Omron CX-Programmer project NewProject (CX-Programmer 9.73)

# PLC PLC_Traffic_Lights: CP1E E20

## Global symbols (name address type ; comment)
0.00 BOOL  ; START
0.01 BOOL  ; STOP
100.00 BOOL  ; LAMPU HIJAU SIMPANG 1
100.01 BOOL  ; LAMPU KUNING SIMPANG 1
100.02 BOOL  ; LAMPU MERAH SIMPANG 1
100.03 BOOL  ; LAMPU HIJAU SIMPANG 2
100.04 BOOL  ; LAMPU KUNING SIMPANG 2
100.05 BOOL  ; LAMPU MERAH SIMPANG 2
100.06 BOOL  ; LAMPU HIJAU SIMPANG 3
100.07 BOOL  ; LAMPU KUNING SIMPANG 3
100.08 BOOL  ; LAMPU MERAH SIMPANG 3
100.09 BOOL  ; LAMPU HIJAU SIMPANG 4
100.10 BOOL  ; LAMPU KUNING SIMPANG 4
100.11 BOOL  ; LAMPU MERAH SIMPANG 4
100.12 BOOL  ; LAMPU PEJALAN KAKI MERAH 1
100.13 BOOL  ; LAMPU PEJALAN KAKI MERAH 2
100.14 BOOL  ; LAMPU PEJALAN KAKI MERAH 3
100.15 BOOL  ; LAMPU PEJALAN KAKI MERAH 4
101.00 BOOL  ; LAMPU PEJALAN KAKI MERAH 1
101.01 BOOL  ; LAMPU PEJALAN KAKI HIJAU 1
101.02 BOOL  ; LAMPU PEJALAN KAKI MERAH 2
101.03 BOOL  ; LAMPU PEJALAN KAKI HIJAU 2
101.04 BOOL  ; LAMPU PEJALAN KAKI MERAH 3
101.05 BOOL  ; LAMPU PEJALAN KAKI HIJAU 3
101.06 BOOL  ; LAMPU PEJALAN KAKI MERAH 3
101.07 BOOL  ; LAMPU PEJALAN KAKI HIJAU 4
99.00 BOOL  ; LAMPU PEJALAN KAKI HIJAU 1
99.01 BOOL  ; LAMPU PEJALAN KAKI HIJAU 2
99.02 BOOL  ; LAMPU PEJALAN KAKI HIJAU 3
99.03 BOOL  ; LAMPU PEJALAN KAKI HIJAU 4
W0.00 BOOL  ; RUNNING

## Program NewProgram1 (cyclic task 0)
; PLC Traffic Lights

### Section Section1

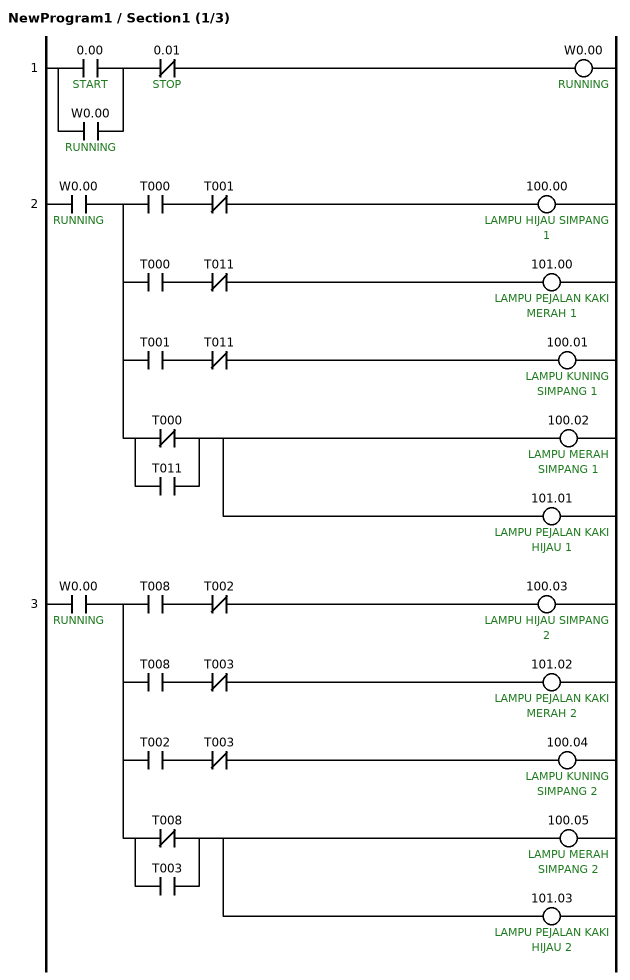
; rung 1
LD 0.00  ; START
OR W0.00  ; RUNNING
ANDNOT 0.01  ; STOP
OUT W0.00  ; RUNNING
; rung 2
LD W0.00  ; RUNNING
OUT TR0
AND T000
ANDNOT T001
OUT 100.00  ; LAMPU HIJAU SIMPANG 1
LD TR0
AND T000
ANDNOT T011
OUT 101.00  ; LAMPU PEJALAN KAKI MERAH 1
LD TR0
AND T001
ANDNOT T011
OUT 100.01  ; LAMPU KUNING SIMPANG 1
LD TR0
LDNOT T000
OR T011
ANDLD
OUT 100.02  ; LAMPU MERAH SIMPANG 1
OUT 101.01  ; LAMPU PEJALAN KAKI HIJAU 1
; rung 3
LD W0.00  ; RUNNING
OUT TR0
AND T008
ANDNOT T002
OUT 100.03  ; LAMPU HIJAU SIMPANG 2
LD TR0
AND T008
ANDNOT T003
OUT 101.02  ; LAMPU PEJALAN KAKI MERAH 2
LD TR0
AND T002
ANDNOT T003
OUT 100.04  ; LAMPU KUNING SIMPANG 2
LD TR0
LDNOT T008
OR T003
ANDLD
OUT 100.05  ; LAMPU MERAH SIMPANG 2
OUT 101.03  ; LAMPU PEJALAN KAKI HIJAU 2

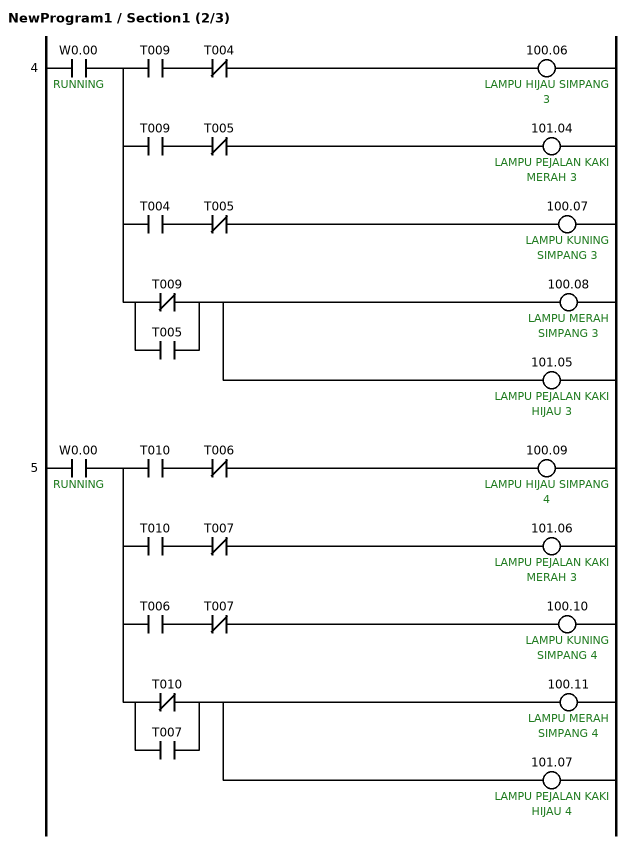
; rung 4
LD W0.00  ; RUNNING
OUT TR0
AND T009
ANDNOT T004
OUT 100.06  ; LAMPU HIJAU SIMPANG 3
LD TR0
AND T009
ANDNOT T005
OUT 101.04  ; LAMPU PEJALAN KAKI MERAH 3
LD TR0
AND T004
ANDNOT T005
OUT 100.07  ; LAMPU KUNING SIMPANG 3
LD TR0
LDNOT T009
OR T005
ANDLD
OUT 100.08  ; LAMPU MERAH SIMPANG 3
OUT 101.05  ; LAMPU PEJALAN KAKI HIJAU 3
; rung 5
LD W0.00  ; RUNNING
OUT TR0
AND T010
ANDNOT T006
OUT 100.09  ; LAMPU HIJAU SIMPANG 4
LD TR0
AND T010
ANDNOT T007
OUT 101.06  ; LAMPU PEJALAN KAKI MERAH 3
LD TR0
AND T006
ANDNOT T007
OUT 100.10  ; LAMPU KUNING SIMPANG 4
LD TR0
LDNOT T010
OR T007
ANDLD
OUT 100.11  ; LAMPU MERAH SIMPANG 4
OUT 101.07  ; LAMPU PEJALAN KAKI HIJAU 4

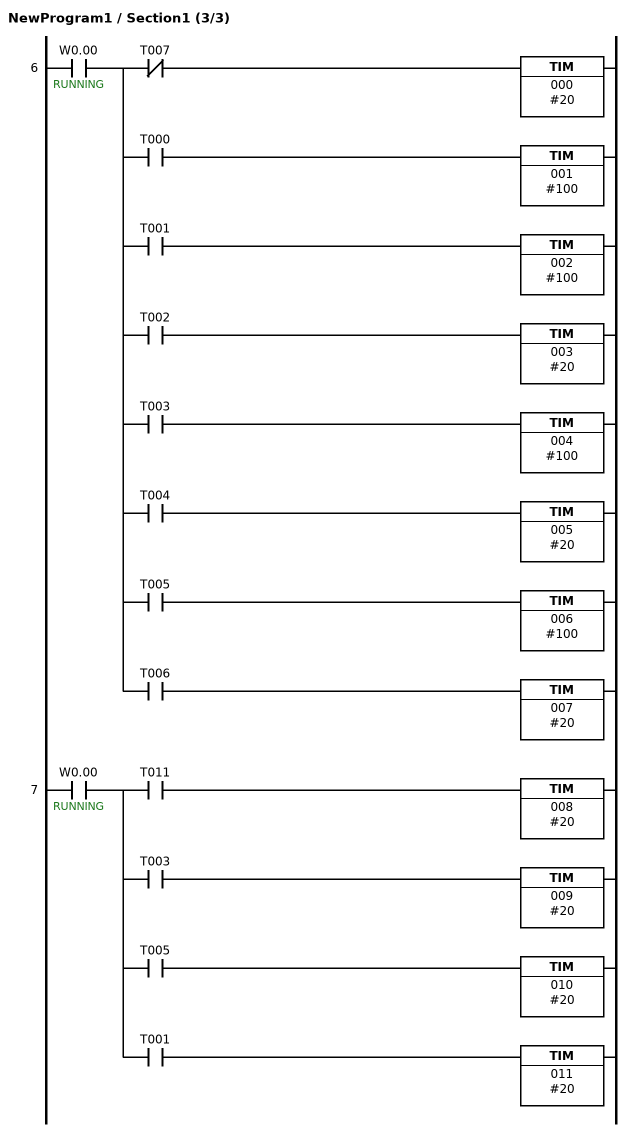
; rung 6
LD W0.00  ; RUNNING
OUT TR0
ANDNOT T007
TIM 000 #20
LD TR0
AND T000
TIM 001 #100
LD TR0
AND T001
TIM 002 #100
LD TR0
AND T002
TIM 003 #20
LD TR0
AND T003
TIM 004 #100
LD TR0
AND T004
TIM 005 #20
LD TR0
AND T005
TIM 006 #100
LD TR0
AND T006
TIM 007 #20
; rung 7
LD W0.00  ; RUNNING
OUT TR0
AND T011
TIM 008 #20
LD TR0
AND T003
TIM 009 #20
LD TR0
AND T005
TIM 010 #20
LD TR0
AND T001
TIM 011 #20

### Section END
; rung 0
END(001)